(* IEC 61131-3 sources: Std_PalletMover/Class/CanOpenWewoBase, 1 file *)

(* ---- CanOpenWewoBase.st ---- *)
(*!
<Class
	Name               = "CanOpenWewoBase"
	Revision           = "0.1"
	RealtimeTask       = "false"
	CyclicTask         = "true"
	DefCyclictime      = "1 ms"
	BackgroundTask     = "false"
	Sigmatek           = "false"
	OSInterface        = "false"
	HighPriority       = "false"
	Automatic          = "false"
	UpdateMode         = "Prescan"
	SharedCommandTable = "true"
	Objectsize         = "(540,240)">
	<Channels>
	</Channels>
	<RevDoku>
		<Owner Company="Riwo Engineering B.V." Author="A.J. Mensink"/>
		<Dokumentation Revision="0.1" Date="2014-03-07" Author="A.J. Mensink" Company="Riwo Engineering B.V." Description="Added new variable: TxDataRiwo"/>
		<Dokumentation Revision="0.0" Date="2014-03-07" Author="A.J. Mensink" Company="Riwo Engineering B.V." Description="First Creation"/>
	</RevDoku>
	<Network Name="CanOpenWewoBase">
		<!-- List of Components in this network -->
		<Components>
			<Object
				Name       = "_base"
				Class      = "CanOpenBase"
				Position   = "(218,120)"
				Visualized = "true">
				<Channels>
					<Server Name="Server0"/>
					<Client Name="cNode"/>
					<Client Name="ConfigData"/>
					<Client Name="Driver"/>
				</Channels>
			</Object>
		</Components>
		<Comments>
		</Comments>
		<!-- List of Connections in this network -->
		<Connections>
			<Connection Source="this.Server0" Destination="_base.Server0" Vertices="(946,210),(774,210),"/>
			<Connection Source="_base.Driver" Destination="this.Driver" Vertices="(218,210),(38,210),"/>
			<Connection Source="_base.cNode" Destination="this.cNode" Vertices="(218,270),(38,270),"/>
			<Connection Source="_base.ConfigData" Destination="this.ConfigData" Vertices="(218,330),(38,330),"/>
		</Connections>
		<!-- Headerfiles -->
		<Options>
		</Options>
	</Network>
</Class>
*)
#pragma using CanOpenBase

CanOpenWewoBase : CLASS
: CanOpenBase
  //Servers:
  //Clients:
  //Variables:
		CanTxData 	: CanObjStr;
  //Functions:

	FUNCTION GLOBAL SendPDO
		VAR_INPUT
			PdoId 	: HINT;
			Bytes 	: BYTE;
			Value1 	: INT;
			Value2 	: INT;
			Value3 	: INT;
			Value4 	: INT;
		END_VAR
		VAR_OUTPUT
			State 	: DINT;
		END_VAR;

	FUNCTION GLOBAL GetPDO
		VAR_INPUT
			PdoId 	: HINT;
		END_VAR
		VAR_OUTPUT
			pCanData 	: ^CanObjStr;
		END_VAR;
  //Tables:
	FUNCTION @STD
		VAR_OUTPUT
			ret_code	: CONFSTATES;
		END_VAR;
	FUNCTION GLOBAL TAB @CT_;
END_CLASS;

FUNCTION GLOBAL CanOpenWewoBase::SendPDO
	VAR_INPUT
		PdoId 	: HINT;
		Bytes 	: BYTE;
		Value1 	: INT;
		Value2 	: INT;
		Value3 	: INT;
		Value4 	: INT;
	END_VAR
	VAR_OUTPUT
		State 	: DINT;
	END_VAR

     // send object
    CanTxData.Id			        := PdoId + to_uint(cNode);
    CanTxData.Size			    := Bytes;
    CanTxData.Data[1]$Int	:= Value1;
    CanTxData.Data[3]$Int	:= Value2;
    CanTxData.Data[5]$Int	:= Value3;
    CanTxData.Data[7]$Int	:= Value4;

    State	:= SendCanObj( #CanTxData);
    If State>= 0 Then
      tPdoSend	:= Ops.tAbsolute;
    End_If;

END_FUNCTION

FUNCTION GLOBAL CanOpenWewoBase::GetPDO
	VAR_INPUT
		PdoId 	: HINT;
	END_VAR
	VAR_OUTPUT
		pCanData 	: ^CanObjStr;
	END_VAR

    pCanData := GetCanObj( ObjNr:=( PdoId + To_Uint( cNode)));

END_FUNCTION
